{attribute 'GeneratedUsingTerminal: EL5151-0000-0020'}
{attribute addProperty BoxType "EL5151-0000-0020"}
{attribute addProperty Id "EtcSlaveTerminalBaseENC_InputsAT %I*ENC_Inputs_B353648514ENC_Inputs_1AT %I*ENC_Inputs_24B63C534ENC_OutputsAT %Q*ENC_Outputs_21E2D14D6WcStateAT %I*WcState_9091E0EB2InfoDataAT %I*InfoData_32EB74EA10"}
{attribute addProperty CRC "647865711"}
{attribute addProperty Size "36"}
TYPE EL5151_269DA56F EXTENDS EtcSlaveTerminalBase :
STRUCT
	{attribute addProperty Name "ENC_Inputs"}
	ENC_Inputs : ENC_Inputs_B3536485;
	{attribute addProperty Name "ENC_Inputs_1"}
	ENC_Inputs_1 : ENC_Inputs_24B63C53;
	{attribute addProperty Name "ENC_Outputs"}
	ENC_Outputs : ENC_Outputs_21E2D14D;
	{attribute addProperty Name "WcState"}
	WcState : WcState_9091E0EB;
	{attribute addProperty Name "InfoData"}
	InfoData : InfoData_32EB74EA;
END_STRUCT
END_TYPE

(* stored: Version 1.2.0.0, ProductVersion 3.1.4024.9
   DUT EL5151_269DA56F: Id {e532c472-8abb-42fb-982d-0f7916cc41f2} *)
